// TwinCAT 3 PLC project SolidAttenuatorPLC
// ProgramVersion: 3.1.4022.7
// libraries:
//   lcls-twincat-motion, * (SLAC)
//   Tc2_Standard, * (Beckhoff Automation GmbH)
//   Tc2_System, * (Beckhoff Automation GmbH)
//   Tc3_Module, * (Beckhoff Automation GmbH)
//   LCLS General,0.0.0,SLAC
// project tree:
//   GVLs/ Main.TcGVL
//   / PlcTask.TcTTO (not stored)
//   POUs/ PRG_1_PlcTask.TcPOU, FB_SATT.TcPOU, PRG_2_AT1K4.TcPOU
// real-time tasks:
//   TASK PlcTask: cycle T#10ms, priority 20, ADS port 350
// motion (NC):
// I/O:
//   DEVICE Device 3 (EtherCAT), AmsNetId 192.168.58.1.4.1
//     Term 1 (EK1100) [EK1100 EtherCAT Coupler (2A E-Bus)]
//       AT1K4-EL7047-01 [EL7047 1Ch. Stepper motor output stage (50V, 5A)]
//       AT1K4-EL7047-02 [EL7047 1Ch. Stepper motor output stage (50V, 5A)]
//       AT1K4-EL7047-03 [EL7047 1Ch. Stepper motor output stage (50V, 5A)]
//       AT1K4-EL7047-04 [EL7047 1Ch. Stepper motor output stage (50V, 5A)]
//       AT1K4-EL5042-01 [EL5042 2Ch. BiSS-C Encoder]
//       AT1K4-EL5042-02 [EL5042 2Ch. BiSS-C Encoder]
//       AT1K4-EL3202-01 [EL3202-0020 2Ch. Ana. Input PT100 (RTD), High Precision, calibrated]
//       AT1K4-EL3202-02 [EL3202-0020 2Ch. Ana. Input PT100 (RTD), High Precision, calibrated]
//       AT1K4-EL3202-03 [EL3202-0020 2Ch. Ana. Input PT100 (RTD), High Precision, calibrated]
//       AT1K4-EL3202-04 [EL3202-0020 2Ch. Ana. Input PT100 (RTD), High Precision, calibrated]
//       Term 12 (EL9011) [EL9011 End Terminal]
// variable links:
//   SolidAttenuatorPLC Instance <-> Device 3 (EtherCAT)/Term 1 (EK1100)/AT1K4-EL3202-01
//     PlcTask Inputs/PRG_2_AT1K4.prg_2_at1k4.RTD_Axis1_1.bError <-> RTD Inputs Channel 1/Status/Error
//     PlcTask Inputs/PRG_2_AT1K4.prg_2_at1k4.RTD_Axis1_2.bError <-> RTD Inputs Channel 2/Status/Error
//     PlcTask Inputs/PRG_2_AT1K4.prg_2_at1k4.RTD_Axis1_1.bOverrange <-> RTD Inputs Channel 1/Status/Overrange
//     PlcTask Inputs/PRG_2_AT1K4.prg_2_at1k4.RTD_Axis1_2.bOverrange <-> RTD Inputs Channel 2/Status/Overrange
//     PlcTask Inputs/PRG_2_AT1K4.prg_2_at1k4.RTD_Axis1_1.bUnderrange <-> RTD Inputs Channel 1/Status/Underrange
//     PlcTask Inputs/PRG_2_AT1K4.prg_2_at1k4.RTD_Axis1_2.bUnderrange <-> RTD Inputs Channel 2/Status/Underrange
//     PlcTask Inputs/PRG_2_AT1K4.prg_2_at1k4.RTD_Axis1_1.iRaw <-> RTD Inputs Channel 1/Value
//     PlcTask Inputs/PRG_2_AT1K4.prg_2_at1k4.RTD_Axis1_2.iRaw <-> RTD Inputs Channel 2/Value
//   SolidAttenuatorPLC Instance <-> Device 3 (EtherCAT)/Term 1 (EK1100)/AT1K4-EL3202-02
//     PlcTask Inputs/PRG_2_AT1K4.prg_2_at1k4.RTD_Axis2_1.bError <-> RTD Inputs Channel 1/Status/Error
//     PlcTask Inputs/PRG_2_AT1K4.prg_2_at1k4.RTD_Axis2_2.bError <-> RTD Inputs Channel 2/Status/Error
//     PlcTask Inputs/PRG_2_AT1K4.prg_2_at1k4.RTD_Axis2_1.bOverrange <-> RTD Inputs Channel 1/Status/Overrange
//     PlcTask Inputs/PRG_2_AT1K4.prg_2_at1k4.RTD_Axis2_2.bOverrange <-> RTD Inputs Channel 2/Status/Overrange
//     PlcTask Inputs/PRG_2_AT1K4.prg_2_at1k4.RTD_Axis2_1.bUnderrange <-> RTD Inputs Channel 1/Status/Underrange
//     PlcTask Inputs/PRG_2_AT1K4.prg_2_at1k4.RTD_Axis2_2.bUnderrange <-> RTD Inputs Channel 2/Status/Underrange
//     PlcTask Inputs/PRG_2_AT1K4.prg_2_at1k4.RTD_Axis2_1.iRaw <-> RTD Inputs Channel 1/Value
//     PlcTask Inputs/PRG_2_AT1K4.prg_2_at1k4.RTD_Axis2_2.iRaw <-> RTD Inputs Channel 2/Value
//   SolidAttenuatorPLC Instance <-> Device 3 (EtherCAT)/Term 1 (EK1100)/AT1K4-EL3202-03
//     PlcTask Inputs/PRG_2_AT1K4.prg_2_at1k4.RTD_Axis3_1.bError <-> RTD Inputs Channel 1/Status/Error
//     PlcTask Inputs/PRG_2_AT1K4.prg_2_at1k4.RTD_Axis3_2.bError <-> RTD Inputs Channel 2/Status/Error
//     PlcTask Inputs/PRG_2_AT1K4.prg_2_at1k4.RTD_Axis3_1.bOverrange <-> RTD Inputs Channel 1/Status/Overrange
//     PlcTask Inputs/PRG_2_AT1K4.prg_2_at1k4.RTD_Axis3_2.bOverrange <-> RTD Inputs Channel 2/Status/Overrange
//     PlcTask Inputs/PRG_2_AT1K4.prg_2_at1k4.RTD_Axis3_1.bUnderrange <-> RTD Inputs Channel 1/Status/Underrange
//     PlcTask Inputs/PRG_2_AT1K4.prg_2_at1k4.RTD_Axis3_2.bUnderrange <-> RTD Inputs Channel 2/Status/Underrange
//     PlcTask Inputs/PRG_2_AT1K4.prg_2_at1k4.RTD_Axis3_1.iRaw <-> RTD Inputs Channel 1/Value
//     PlcTask Inputs/PRG_2_AT1K4.prg_2_at1k4.RTD_Axis3_2.iRaw <-> RTD Inputs Channel 2/Value
//   SolidAttenuatorPLC Instance <-> Device 3 (EtherCAT)/Term 1 (EK1100)/AT1K4-EL3202-04
//     PlcTask Inputs/PRG_2_AT1K4.prg_2_at1k4.RTD_Axis4_1.bError <-> RTD Inputs Channel 1/Status/Error
//     PlcTask Inputs/PRG_2_AT1K4.prg_2_at1k4.RTD_Axis4_2.bError <-> RTD Inputs Channel 2/Status/Error
//     PlcTask Inputs/PRG_2_AT1K4.prg_2_at1k4.RTD_Axis4_1.bOverrange <-> RTD Inputs Channel 1/Status/Overrange
//     PlcTask Inputs/PRG_2_AT1K4.prg_2_at1k4.RTD_Axis4_2.bOverrange <-> RTD Inputs Channel 2/Status/Overrange
//     PlcTask Inputs/PRG_2_AT1K4.prg_2_at1k4.RTD_Axis4_1.bUnderrange <-> RTD Inputs Channel 1/Status/Underrange
//     PlcTask Inputs/PRG_2_AT1K4.prg_2_at1k4.RTD_Axis4_2.bUnderrange <-> RTD Inputs Channel 2/Status/Underrange
//     PlcTask Inputs/PRG_2_AT1K4.prg_2_at1k4.RTD_Axis4_1.iRaw <-> RTD Inputs Channel 1/Value
//     PlcTask Inputs/PRG_2_AT1K4.prg_2_at1k4.RTD_Axis4_2.iRaw <-> RTD Inputs Channel 2/Value
//   SolidAttenuatorPLC Instance <-> Device 3 (EtherCAT)/Term 1 (EK1100)/AT1K4-EL7047-01
//     PlcTask Inputs/Main.M1.bLimitBackwardEnable <-> STM Status/Status/Digital input 2
//     PlcTask Inputs/Main.M1.bLimitForwardEnable <-> STM Status/Status/Digital input 1
//   SolidAttenuatorPLC Instance <-> Device 3 (EtherCAT)/Term 1 (EK1100)/AT1K4-EL7047-02
//     PlcTask Inputs/Main.M2.bLimitBackwardEnable <-> STM Status/Status/Digital input 2
//     PlcTask Inputs/Main.M2.bLimitForwardEnable <-> STM Status/Status/Digital input 1
//   SolidAttenuatorPLC Instance <-> Device 3 (EtherCAT)/Term 1 (EK1100)/AT1K4-EL7047-03
//     PlcTask Inputs/Main.M3.bLimitBackwardEnable <-> STM Status/Status/Digital input 2
//     PlcTask Inputs/Main.M3.bLimitForwardEnable <-> STM Status/Status/Digital input 1
//   SolidAttenuatorPLC Instance <-> Device 3 (EtherCAT)/Term 1 (EK1100)/AT1K4-EL7047-04
//     PlcTask Inputs/Main.M4.bLimitBackwardEnable <-> STM Status/Status/Digital input 2
//     PlcTask Inputs/Main.M4.bLimitForwardEnable <-> STM Status/Status/Digital input 1
//   SolidAttenuatorPLC Instance <-> NC-Task 1 SAF/Axes/AT1K4-M1
//     PlcTask Inputs/Main.M1.Axis.NcToPlc <-> Outputs/ToPlc
//     PlcTask Outputs/Main.M1.Axis.PlcToNc <-> Inputs/FromPlc
//   SolidAttenuatorPLC Instance <-> NC-Task 1 SAF/Axes/AT1K4-M2
//     PlcTask Inputs/Main.M2.Axis.NcToPlc <-> Outputs/ToPlc
//     PlcTask Outputs/Main.M2.Axis.PlcToNc <-> Inputs/FromPlc
//   SolidAttenuatorPLC Instance <-> NC-Task 1 SAF/Axes/AT1K4-M3
//     PlcTask Inputs/Main.M3.Axis.NcToPlc <-> Outputs/ToPlc
//     PlcTask Outputs/Main.M3.Axis.PlcToNc <-> Inputs/FromPlc
//   SolidAttenuatorPLC Instance <-> NC-Task 1 SAF/Axes/AT1K4-M4
//     PlcTask Inputs/Main.M4.Axis.NcToPlc <-> Outputs/ToPlc
//     PlcTask Outputs/Main.M4.Axis.PlcToNc <-> Inputs/FromPlc

// ---- GVLs/Main.TcGVL
{attribute 'qualified_only'}
VAR_GLOBAL
(*
    Only includes motor definitions for the IOC
    These are hard-coded to be Main.M#,
    but are very convenient to store in a GVL,
    hence the confusing namespace here

    This should be refactored once the IOC
    supports arbitrary ads paths for motors
*)
(*
    Four identical systems:
    Instr.		Area		ID#			Z (m)
    TMO			FEE			AT1K4-SOLID	748
    NEH 2.2		H2.2		AT1K2-SOLID	784
    NEH 2.2		H2.2		AT2K2-SOLID	788.8
    TXI			H1.1		AT1K3-SOLID	~763

*)
    {attribute 'pytmc' := 'pv: AT1K4:L2SI:MMS:01'}
    {attribute 'TcLinkTo' := '
        .bLimitForwardEnable  := TIIB[AT1K4-EL7047-01]^STM Status^Status^Digital input 1;
        .bLimitBackwardEnable := TIIB[AT1K4-EL7047-01]^STM Status^Status^Digital input 2;
		.nRawEncoderULINT     := TIIB[AT1K4-EL5042-01]^FB Inputs Channel 1^Position'}
    M1: DUT_MotionStage := (sName := 'AT1K4:L2SI:MMS:01');

    {attribute 'pytmc' := 'pv: AT1K4:L2SI:MMS:02'}
    {attribute 'TcLinkTo' := '
        .bLimitForwardEnable  := TIIB[AT1K4-EL7047-02]^STM Status^Status^Digital input 1;
        .bLimitBackwardEnable := TIIB[AT1K4-EL7047-02]^STM Status^Status^Digital input 2;
		.nRawEncoderULINT     := TIIB[AT1K4-EL5042-01]^FB Inputs Channel 2^Position'}
    
    M2: DUT_MotionStage := (sName := 'AT1K4:L2SI:MMS:02');

    {attribute 'pytmc' := 'pv: AT1K4:L2SI:MMS:03'}
    {attribute 'TcLinkTo' := '
        .bLimitForwardEnable  := TIIB[AT1K4-EL7047-03]^STM Status^Status^Digital input 1;
        .bLimitBackwardEnable := TIIB[AT1K4-EL7047-03]^STM Status^Status^Digital input 2;
		.nRawEncoderULINT     := TIIB[AT1K4-EL5042-02]^FB Inputs Channel 1^Position'}
    
    M3: DUT_MotionStage := (sName := 'AT1K4:L2SI:MMS:03');

    {attribute 'pytmc' := 'pv: AT1K4:L2SI:MMS:04'}
    {attribute 'TcLinkTo' := '
        .bLimitForwardEnable  := TIIB[AT1K4-EL7047-04]^STM Status^Status^Digital input 1;
        .bLimitBackwardEnable := TIIB[AT1K4-EL7047-04]^STM Status^Status^Digital input 2;
		.nRawEncoderULINT     := TIIB[AT1K4-EL5042-02]^FB Inputs Channel 1^Position'}
    M4: DUT_MotionStage := (sName := 'AT1K4:L2SI:MMS:04');

END_VAR

// ---- POUs/PRG_1_PlcTask.TcPOU

PROGRAM PRG_1_PlcTask
VAR
    fbLogHandler: FB_LogHandler;

 

END_VAR

fbLogHandler();


PRG_2_AT1K4();

END_PROGRAM

// ---- POUs/PRG_2_AT1K4.TcPOU
PROGRAM PRG_2_AT1K4
VAR
	
   {attribute 'pytmc' := 'pv: AT1K4:L2SI:'}
    {attribute 'TcLinkTo' := '
        .RTD_Axis1_1.iRaw := TIIB[AT1K4-EL3202-01]^RTD Inputs Channel 1^Value;
        .RTD_Axis1_1.bError := TIIB[AT1K4-EL3202-01]^RTD Inputs Channel 1^Status^Error;
        .RTD_Axis1_1.bUnderrange := TIIB[AT1K4-EL3202-01]^RTD Inputs Channel 1^Status^Underrange;
        .RTD_Axis1_1.bOverrange := TIIB[AT1K4-EL3202-01]^RTD Inputs Channel 1^Status^Overrange;

        .RTD_Axis1_2.iRaw := TIIB[AT1K4-EL3202-01]^RTD Inputs Channel 2^Value;
        .RTD_Axis1_2.bError := TIIB[AT1K4-EL3202-01]^RTD Inputs Channel 2^Status^Error;
        .RTD_Axis1_2.bUnderrange := TIIB[AT1K4-EL3202-01]^RTD Inputs Channel 2^Status^Underrange;
        .RTD_Axis1_2.bOverrange := TIIB[AT1K4-EL3202-01]^RTD Inputs Channel 2^Status^Overrange;


        .RTD_Axis2_1.iRaw := TIIB[AT1K4-EL3202-02]^RTD Inputs Channel 1^Value;
        .RTD_Axis2_1.bError := TIIB[AT1K4-EL3202-02]^RTD Inputs Channel 1^Status^Error;
        .RTD_Axis2_1.bUnderrange := TIIB[AT1K4-EL3202-02]^RTD Inputs Channel 1^Status^Underrange;
        .RTD_Axis2_1.bOverrange := TIIB[AT1K4-EL3202-02]^RTD Inputs Channel 1^Status^Overrange;

        .RTD_Axis2_2.iRaw := TIIB[AT1K4-EL3202-02]^RTD Inputs Channel 2^Value;
        .RTD_Axis2_2.bError := TIIB[AT1K4-EL3202-02]^RTD Inputs Channel 2^Status^Error;
        .RTD_Axis2_2.bUnderrange := TIIB[AT1K4-EL3202-02]^RTD Inputs Channel 2^Status^Underrange;
        .RTD_Axis2_2.bOverrange := TIIB[AT1K4-EL3202-02]^RTD Inputs Channel 2^Status^Overrange;


        .RTD_Axis3_1.iRaw := TIIB[AT1K4-EL3202-03]^RTD Inputs Channel 1^Value;
        .RTD_Axis3_1.bError := TIIB[AT1K4-EL3202-03]^RTD Inputs Channel 1^Status^Error;
        .RTD_Axis3_1.bUnderrange := TIIB[AT1K4-EL3202-03]^RTD Inputs Channel 1^Status^Underrange;
        .RTD_Axis3_1.bOverrange := TIIB[AT1K4-EL3202-03]^RTD Inputs Channel 1^Status^Overrange;

        .RTD_Axis3_2.iRaw := TIIB[AT1K4-EL3202-03]^RTD Inputs Channel 2^Value;
        .RTD_Axis3_2.bError := TIIB[AT1K4-EL3202-03]^RTD Inputs Channel 2^Status^Error;
        .RTD_Axis3_2.bUnderrange := TIIB[AT1K4-EL3202-03]^RTD Inputs Channel 2^Status^Underrange;
        .RTD_Axis3_2.bOverrange := TIIB[AT1K4-EL3202-03]^RTD Inputs Channel 2^Status^Overrange;


        .RTD_Axis4_1.iRaw := TIIB[AT1K4-EL3202-04]^RTD Inputs Channel 1^Value;
        .RTD_Axis4_1.bError := TIIB[AT1K4-EL3202-04]^RTD Inputs Channel 1^Status^Error;
        .RTD_Axis4_1.bUnderrange := TIIB[AT1K4-EL3202-04]^RTD Inputs Channel 1^Status^Underrange;
        .RTD_Axis4_1.bOverrange := TIIB[AT1K4-EL3202-04]^RTD Inputs Channel 1^Status^Overrange;

        .RTD_Axis4_2.iRaw := TIIB[AT1K4-EL3202-04]^RTD Inputs Channel 2^Value;
        .RTD_Axis4_2.bError := TIIB[AT1K4-EL3202-04]^RTD Inputs Channel 2^Status^Error;
        .RTD_Axis4_2.bUnderrange := TIIB[AT1K4-EL3202-04]^RTD Inputs Channel 2^Status^Underrange;
        .RTD_Axis4_2.bOverrange := TIIB[AT1K4-EL3202-04]^RTD Inputs Channel 2^Status^Overrange;

    '}
    prg_2_at1k4 : FB_SATT;
	
	 bDebug : BOOL := FALSE;
    nEnableMode: ENUM_StageEnableMode;
	
END_VAR

(* Motion *)

IF bDebug THEN
    // NEVER: checkouts with the TwinCAT NC GUI.
    nEnableMode := ENUM_StageEnableMode.NEVER;
ELSE
    // ALWAYS: want active position correction at all times
    nEnableMode := ENUM_StageEnableMode.ALWAYS;
END_IF


prg_2_at1k4(stMotion1:=Main.M1,
			stMotion2:=Main.M2,
			stMotion3:=Main.M3,
			stMotion4:=Main.M4,
			nEnableMode:= nEnableMode);

END_PROGRAM

// ---- POUs/FB_SATT.TcPOU
FUNCTION_BLOCK FB_SATT
VAR_INPUT
	stMotion1: DUT_MotionStage;
	stMotion2: DUT_MotionStage;
	stMotion3: DUT_MotionStage;
	stMotion4: DUT_MotionStage;
	nEnableMode: ENUM_StageEnableMode;
END_VAR
VAR_OUTPUT
END_VAR
VAR
 
    (*
        The 4 motion axes - linked to GVL Main.{M1, M2, M3, and M4}.

        Note that the DUT_MotionStage is where the pytmc pragmas go.
    *)
	fbMotion1: FB_MotionStage;
    fbMotion2: FB_MotionStage;
    fbMotion3: FB_MotionStage;
    fbMotion4: FB_MotionStage;
  

    (* EL3202-0020: 0.01 °C per digit *)
    {attribute 'pytmc' := 'pv: MMS:01:RTD1'}
    RTD_Axis1_1: FB_TempSensor := ( fResolution:=0.01 );
    {attribute 'pytmc' := 'pv: MMS:01:RTD2'}
    RTD_Axis1_2: FB_TempSensor := ( fResolution:=0.01 );

    {attribute 'pytmc' := 'pv: MMS:02:RTD1'}
    RTD_Axis2_1: FB_TempSensor := ( fResolution:=0.01 );
    {attribute 'pytmc' := 'pv: MMS:02:RTD2'}
    RTD_Axis2_2: FB_TempSensor := ( fResolution:=0.01 );

    {attribute 'pytmc' := 'pv: MMS:03:RTD1'}
    RTD_Axis3_1: FB_TempSensor := ( fResolution:=0.01 );
    {attribute 'pytmc' := 'pv: MMS:03:RTD2'}
    RTD_Axis3_2: FB_TempSensor := ( fResolution:=0.01 );

    {attribute 'pytmc' := 'pv: MMS:04:RTD1'}
    RTD_Axis4_1: FB_TempSensor := ( fResolution:=0.01 );
    {attribute 'pytmc' := 'pv: MMS:04:RTD2'}
    RTD_Axis4_2: FB_TempSensor := ( fResolution:=0.01 );
	
	bInit:BOOL :=TRUE;

END_VAR

(* RTDs *)
RTD_Axis1_1();
RTD_Axis1_2();

RTD_Axis2_1();
RTD_Axis2_2();

RTD_Axis3_1();
RTD_Axis3_2();

RTD_Axis4_1();
RTD_Axis4_2();

if (bInit) THEN
	bINIT:=FALSE;
	stMotion1.bHardwareEnable      := TRUE;
	stMotion1.bLimitBackwardEnable := TRUE;
	stMotion1.bLimitForwardEnable  := TRUE;
	stMotion1.bPowerSelf           := TRUE;
	stMotion1.nBrakeMode           := ENUM_StageBrakeMode.NO_BRAKE;
	stMotion1.nEnableMode          := nEnableMode;
	stMotion1.nHomingMode          := ENUM_EpicsHomeCmd.NONE;


	stMotion2.bHardwareEnable      := TRUE;
	stMotion2.bLimitBackwardEnable := TRUE;
	stMotion2.bLimitForwardEnable  := TRUE;
	stMotion2.bPowerSelf           := TRUE;
	stMotion2.nBrakeMode           := ENUM_StageBrakeMode.NO_BRAKE;
	stMotion2.nEnableMode          := nEnableMode;
	stMotion2.nHomingMode          := ENUM_EpicsHomeCmd.NONE;

	stMotion3.bHardwareEnable      := TRUE;
	stMotion3.bLimitBackwardEnable := TRUE;
	stMotion3.bLimitForwardEnable  := TRUE;
	stMotion3.bPowerSelf           := TRUE;
	stMotion3.nBrakeMode           := ENUM_StageBrakeMode.NO_BRAKE;
	stMotion3.nEnableMode          := nEnableMode;
	stMotion3.nHomingMode          := ENUM_EpicsHomeCmd.NONE;


	stMotion4.bHardwareEnable      := TRUE;
	stMotion4.bLimitBackwardEnable := TRUE;
	stMotion4.bLimitForwardEnable  := TRUE;
	stMotion4.bPowerSelf           := TRUE;
	stMotion4.nBrakeMode           := ENUM_StageBrakeMode.NO_BRAKE;
	stMotion4.nEnableMode          := nEnableMode;
	stMotion4.nHomingMode          := ENUM_EpicsHomeCmd.NONE;

END_IF

(* Motion *)
fbMotion1(stMotionStage:=Main.M1);
fbMotion2(stMotionStage:=Main.M2);
fbMotion3(stMotionStage:=Main.M3);
fbMotion4(stMotionStage:=Main.M4);

END_FUNCTION_BLOCK
